(* CODESYS project marcha-paro3 G.project
   CustomField01_name: CustomField01
   CustomField08_name: CustomField08
   CustomField06_name: CustomField06
   Title: ATV_IMC_Template
   CustomField09_name: CustomField09
   CustomField07_name: CustomField07
   CustomField05_name: CustomField05
   CustomField02_name: CustomField02
   Description: This template can be used for a correct interface with the local drive. the MANDATORY_AT_EACH_CYCLE program must be called like it is done in this application.
   CustomField04_name: CustomField04
   CustomField10_name: CustomField10
   Version: 0.0.0.0
   Company: Schneider Electric
   CustomField03_name: CustomField03

Project tree, tasks and I/O mapping:
  MyController : TM241CE24R, Schneider Electric, order no. TM241CE24R, version 4.0.3.8
    application Application
      task MAST (cyclic, interval 20 ms, priority 15, watchdog 100 ms x 1) calls principal
      function HiddenPOU [ST]
      global variables GVL
      program principal [SFC]: Tparo
      visualisation simu
    DI : Digital Inputs, Schneider Electric, version 4.0.3.8
        input  iwDI_IW0 : WORD  // IW0
        input  ibDI_IB1 : BYTE  // IB1
    DQ : Digital Outputs, Schneider Electric, version 4.0.3.8
        output qwDQ_QW0 : WORD  // QW0
        output qbDQ_QB1 : BYTE  // QB1
    Counters : Counters, Schneider Electric, version 4.0.3.8
    Pulse_Generators : Pulse Generators, Schneider Electric, version 4.0.3.8
    Cartridge_1 : Cartridge, Schneider Electric, version 4.0.3.8
    IO_Bus : IO bus - TM3, Schneider Electric, version 4.0.3.8
    COM_Bus : COM bus, Schneider Electric, version 4.0.3.8
    Ethernet_1 : Ethernet Network, Schneider Electric, version 4.0.3.8
    Serial_Line_1 : Serial line, Schneider Electric, version 4.0.3.8
      SoMachine_Network_Manager : SoMachine-Network Manager, Schneider Electric, version 4.0.0.2
    Serial_Line_2 : Serial line, Schneider Electric, version 4.0.3.8
      Modbus_Manager : Modbus Manager, Schneider Electric, version 4.0.0.2
  text list GlobalTextList
*)

// MyController/Application/GVL
VAR_GLOBAL
	// boton de marcha
	marcha: BOOL;
	// boton de paro
	paro: BOOL;
	lampara: BOOL;
END_VAR

// MyController/Application/principal
PROGRAM principal
VAR
END_VAR

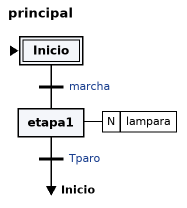
INITIAL_STEP Inicio:
END_STEP
TRANSITION FROM Inicio TO etapa1
    := marcha;
END_TRANSITION
STEP etapa1:
    lampara(N);
END_STEP
TRANSITION FROM etapa1 TO Inicio
    := Tparo;
END_TRANSITION

TRANSITION Tparo:
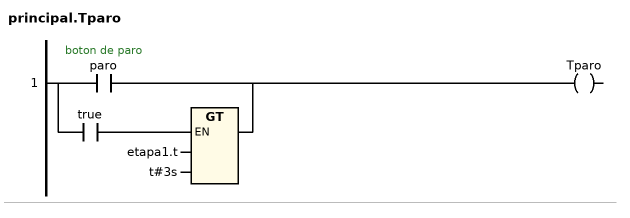
// NETWORK 1
//   paro: boton de paro
Tparo := paro OR true AND etapa1.t > t#3s;
END_TRANSITION

END_PROGRAM

// MyController/Application/HiddenPOU
FUNCTION HiddenPOU : BOOL

VAR_INPUT
	pHiddenFunc: POINTER TO WORD;
END_VAR
VAR
	pRead: POINTER TO BYTE;
	pWrite: POINTER TO BYTE;
END_VAR

pRead := pHiddenFunc + 400;
pWrite := pHiddenFunc + 4400;
HiddenPOU := TRUE;

END_FUNCTION

// MyController/Application/simu
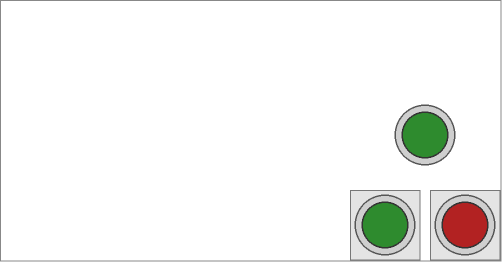
VISUALIZATION simu  // 502x262
    Lamp1 (390,100 70x70), variable: lampara, style: Lamp-Lamp1-Green
    PushSwitch (350,190 70x70), variable: marcha, behaviour: TAP, style: Switch-PushSwitch-Green
    PushSwitch (430,190 70x70), variable: paro, behaviour: TAP, style: Switch-PushSwitch-Red
END_VISUALIZATION
